{attribute 'GeneratedUsingTerminal: EKM1101-0000-0016'}
{attribute addProperty BoxType "EKM1101-0000-0016"}
{attribute addProperty Id "StatusAT %I*Status_BA3D1C5D7Number_of_samplesAT %I*UINT2"}
{attribute addProperty CRC "292982937"}
{attribute addProperty Size "9"}
TYPE MMS_Acceleration_Status_11769099 :
STRUCT
	{attribute addProperty Name "Status"}
	Status AT %I* : Status_BA3D1C5D;
	{attribute addProperty Name "Number_of_samples"}
	Number_of_samples AT %I* : UINT;
END_STRUCT
END_TYPE

(* stored: Version 1.2.0.0, ProductVersion 3.1.4024.9
   DUT MMS_Acceleration_Status_11769099: Id {59799f4c-a90e-4378-8d66-8bbc2d6516bd} *)
